Fanuc TP program (LS listing): test_repo_dst.ls

/PROG  TEST_REPO_DST
/ATTR
OWNER		= MNEDITOR;
COMMENT		= "";
PROG_SIZE	= 1734;
CREATE		= DATE 26-07-23  TIME 17:40:12;
MODIFIED	= DATE 26-07-23  TIME 17:40:12;
FILE_NAME	= TEST_REP;
VERSION		= 0;
LINE_COUNT	= 67;
MEMORY_SIZE	= 2094;
PROTECT		= READ_WRITE;
TCD:  STACK_SIZE	= 0,
      TASK_PRIORITY	= 50,
      TIME_SLICE	= 0,
      BUSY_LAMP_OFF	= 0,
      ABORT_REQUEST	= 0,
      PAUSE_REQUEST	= 0;
DEFAULT_GROUP	= 1,*,*,*,*;
CONTROL_CODE	= 00000000 00000000;
LOCAL_REGISTERS	= 0,0,0;
/APPL
/APPL
/MN
   1:  R[3:REPO_RCP_UOFFSET]=2.799    ;
   2:  R[19:REPO_XOFFSET]=374.85    ;
   3:  R[20:REPO_YOFFSET]=108    ;
   4:  R[21:PICKUP_CONSTANT]=19.5    ;
   5:  R[3:REPO_RCP_UOFFSET]=2.803    ;
   6:   ;
   7:  ! First repo location ;
   8:  PR[5:REPO_RCP_PSN]=P[1:STATIC_REPO_RCP]    ;
   9:  R[48]=R[3:REPO_RCP_UOFFSET]*21    ;
  10:  PR[5,1:REPO_RCP_PSN]=PR[5,1:REPO_RCP_PSN]+R[48]    ;
  11:  R[49]=R[3:REPO_RCP_UOFFSET]*19    ;
  12:  PR[5,2:REPO_RCP_PSN]=PR[5,2:REPO_RCP_PSN]-R[49]    ;
  13:   ;
  14:J P[2:STATIC_HOME] 100% FINE    ;
  15:J PR[5:REPO_RCP_PSN] 100% FINE    ;
  16:   ;
  17:  PR[5,3:REPO_RCP_PSN]=PR[5,3:REPO_RCP_PSN]-R[21:PICKUP_CONSTANT]    ;
  18:   ;
  19:L PR[5:REPO_RCP_PSN] 100mm/sec FINE    ;
  20:   ;
  21:  PR[5,3:REPO_RCP_PSN]=PR[5,3:REPO_RCP_PSN]+R[21:PICKUP_CONSTANT]    ;
  22:   ;
  23:L PR[5:REPO_RCP_PSN] 100mm/sec FINE    ;
  24:   ;
  25:  ! Shift to second repo ;
  26:  PR[5,1:REPO_RCP_PSN]=PR[5,1:REPO_RCP_PSN]+R[19:REPO_XOFFSET]    ;
  27:  PR[5,2:REPO_RCP_PSN]=PR[5,2:REPO_RCP_PSN]-.05    ;
  28:   ;
  29:J PR[5:REPO_RCP_PSN] 100% FINE    ;
  30:   ;
  31:  PR[5,3:REPO_RCP_PSN]=PR[5,3:REPO_RCP_PSN]-R[21:PICKUP_CONSTANT]    ;
  32:   ;
  33:L PR[5:REPO_RCP_PSN] 100mm/sec FINE    ;
  34:   ;
  35:  PR[5,3:REPO_RCP_PSN]=PR[5,3:REPO_RCP_PSN]+R[21:PICKUP_CONSTANT]    ;
  36:   ;
  37:L PR[5:REPO_RCP_PSN] 100mm/sec FINE    ;
  38:   ;
  39:  ! Shift to third repo ;
  40:  PR[5:REPO_RCP_PSN]=P[1:STATIC_REPO_RCP]    ;
  41:  PR[5,1:REPO_RCP_PSN]=PR[5,1:REPO_RCP_PSN]-.1+R[48]    ;
  42:  PR[5,2:REPO_RCP_PSN]=PR[5,2:REPO_RCP_PSN]-R[20:REPO_YOFFSET]-R[49]    ;
  43:   ;
  44:J PR[5:REPO_RCP_PSN] 100% FINE    ;
  45:   ;
  46:  PR[5,3:REPO_RCP_PSN]=PR[5,3:REPO_RCP_PSN]-R[21:PICKUP_CONSTANT]    ;
  47:   ;
  48:L PR[5:REPO_RCP_PSN] 100mm/sec FINE    ;
  49:   ;
  50:  PR[5,3:REPO_RCP_PSN]=PR[5,3:REPO_RCP_PSN]+R[21:PICKUP_CONSTANT]    ;
  51:   ;
  52:L PR[5:REPO_RCP_PSN] 100mm/sec FINE    ;
  53:   ;
  54:  ! Shift to fourth repo ;
  55:  PR[5,1:REPO_RCP_PSN]=PR[5,1:REPO_RCP_PSN]+R[19:REPO_XOFFSET]    ;
  56:  PR[5,2:REPO_RCP_PSN]=PR[5,2:REPO_RCP_PSN]-.05    ;
  57:   ;
  58:J PR[5:REPO_RCP_PSN] 100% FINE    ;
  59:   ;
  60:  PR[5,3:REPO_RCP_PSN]=PR[5,3:REPO_RCP_PSN]-R[21:PICKUP_CONSTANT]    ;
  61:   ;
  62:L PR[5:REPO_RCP_PSN] 100mm/sec FINE    ;
  63:   ;
  64:  PR[5,3:REPO_RCP_PSN]=PR[5,3:REPO_RCP_PSN]+R[21:PICKUP_CONSTANT]    ;
  65:   ;
  66:L PR[5:REPO_RCP_PSN] 100mm/sec FINE    ;
  67:  END ;
/POS
P[1:"STATIC_REPO_RCP"]{
   GP1:
	UF : 1, UT : 1,		CONFIG : 'L, 0, 0, 0',
	X =  -113.481003  mm,	Y =   165.654007  mm,	Z =    15.389000  mm,
	W =   180.000000 deg,	P =     0.000000 deg,	R =     0.000000 deg
};
P[2:"STATIC_HOME"]{
   GP1:
	UF : 1, UT : 1,		CONFIG : 'L, 0, 0, 0',
	X =   100.000000  mm,	Y =   175.000000  mm,	Z =   250.000000  mm,
	W =   180.000000 deg,	P =     0.000000 deg,	R =     0.000000 deg
};
/END
